Universal Robots PolyScope program: comunicacion.urp

Program comunicacion (installation=default directory=/programs createdIn=5.14.5 lastSavedIn=5.14.5 robotSerialNumber=20195300809)
Calibrated DH parameters: a=[-0.000085, -0.20076, -0.212369, 0.000121, -0.000118, 0]; d=[0.15185, -26.306375, 24.753047, 1.684739, 0.085386, 0.092088]; alpha=[1.572149, -0.00522, -0.011864, 1.571339, -1.571085, 0]; deltaTheta=[0, 0.599885, -0.513355, -0.086555, 0.000006, 0]
InitVariablesNode
BeforeStart
  MoveJ speed 60 deg/s, acceleration 80 deg/s^2 (useActiveTCP=true) feature=Base
    Waypoint Waypoint_2: TCP in base x=5.973 y=-372.7 z=694.671 mm, rx=-0.018 ry=2.2102 rz=-2.2165 rad; joints [0.002, -90, -0.002, -90.002, 0, 0.001] deg; TCP offset x=0 y=0 z=150 mm, rx=0 ry=0 rz=0 rad
  abrir := socket_open("10.5.20.90",30003)
  Loop While (checkContinuously=false) expression=abrir≟ False
    Wait Sleep waitTime=0.01
    abrir := socket_open("10.5.20.90",30003)
  tasca := 0
Robot Program (runOnlyOnce=false)
  If tasca≟1
    MoveJ speed 60 deg/s, acceleration 80 deg/s^2 (useActiveTCP=true) feature=Base
      Waypoint Waypoint_1: TCP in base x=-341.363 y=-368.12 z=536.157 mm, rx=0.8414 ry=1.3417 rz=-1.531 rad; joints [-0.182, -70.569, 49.096, -90.536, 10.167, 0.602] deg
    tasca := 0
Thread Thread_1 (runOnlyOnce=false)
  dato := socket_read_ascii_float(1)
  Popup Message (haltProgram=false inputType=Variable) variable=dato
  Loop While (checkContinuously=false) expression=dato[0]≠1
    dato := socket_read_ascii_float(1)
  If dato[1]≟1
    tasca := 1
